# EPICS alarm handler configuration: mps_database/bare/alarms/areas/mpln_sph_mp05.alhConfig
GROUP NULL MPLN:SPH:MP05:1
$ALIAS MPS Link Node 124
$GUIDANCE
LTUH MPS
   Group Name: MPLN:SPH:MP05:1
   Summary PV:  MPLN:SPH:MP05:1:STATSUMY
$END
CHANNEL  MPLN:SPH:MP05:1    MPLN:SPH:MP05:1:MPS_EN_RBV		-----
CHANNEL  MPLN:SPH:MP05:1    MPLN:SPH:MP05:1:LC1_MODE_RBV		-----
